FUNCTION_BLOCK Slider (* Slider for the drill *)
  (* Standard: 61499-2 *)
  (* Version 0.2, 2003-12-04, JHC, Rockwell Automation, Renamed for better indexing. *)
  (* Version 0.1, 2002-11-05, JHC, Rockwell Automation, Corrected missing ST element in Algorithm REQ. *)
  (* Version 0.0, 2000-05-30, JHC, Rockwell Automation *)
  (* Compiler header: package fb.rt.benchmarks.DrillStation; *)
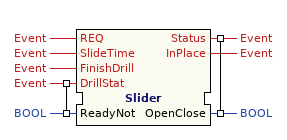
  EVENT_INPUT
    REQ; (* Normal Execution Request *)
    SlideTime; (* Simulate the sliding time *)
    FinishDrill;
    DrillStat WITH ReadyNot; (* Status of the drill *)
  END_EVENT
  EVENT_OUTPUT
    Status WITH OpenClose;
    InPlace; (* Object is in place for drilling *)
  END_EVENT
  VAR_INPUT
    ReadyNot : BOOL; (* ready: true, not ready: false *)
  END_VAR
  VAR_OUTPUT
    OpenClose : BOOL := true; (* true: open, false: close *)
  END_VAR
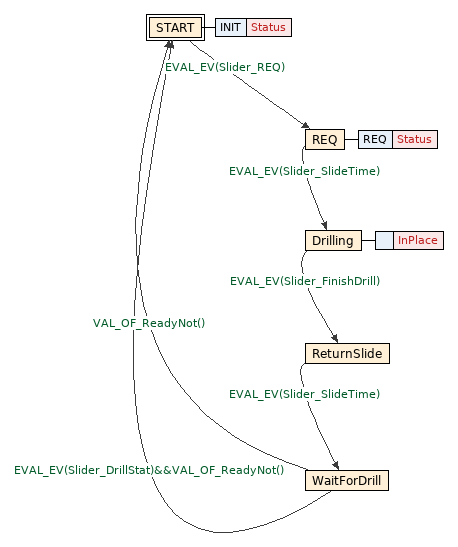
  EC_STATES
    START : INIT -> Status; (* Initial State *)
    REQ : REQ -> Status; (* Normal execution *)
    Drilling : -> InPlace;
    ReturnSlide;
    WaitForDrill;
  END_STATES
  EC_TRANSITIONS
    START TO REQ := EVAL_EV(Slider_REQ);
    REQ TO Drilling := EVAL_EV(Slider_SlideTime);
    Drilling TO ReturnSlide := EVAL_EV(Slider_FinishDrill);
    ReturnSlide TO WaitForDrill := EVAL_EV(Slider_SlideTime);
    WaitForDrill TO START := VAL_OF_ReadyNot();
    WaitForDrill TO START := EVAL_EV(Slider_DrillStat)&&VAL_OF_ReadyNot();
  END_TRANSITIONS
  ALGORITHM INIT IN ST: (* Initialization algorithm *)
VAL_OF_OpenClose() = 1;
  END_ALGORITHM
  ALGORITHM REQ IN ST: (* Normally executed algorithm *)
VAL_OF_OpenClose() = 0;
  END_ALGORITHM
END_FUNCTION_BLOCK
